Yaskawa INFORM job: FRONT_WELD_-90ST-1_5340.JBI

/JOB
//NAME FRONT_WELD_-90ST-1_5340
///FOLDERNAME 02-SKRZYNIE_JOBS
//POS
///NPOS 21,21,0,4,0,0
///TOOL 0
///POSTYPE PULSE
///PULSE
C00000=0,-52278,40443,0,6873,1
C00001=0,-52278,40443,0,6873,-1
C00002=0,-52278,40443,-5610,-49281,70968
C00003=0,-42686,23640,-7425,-34877,79161
C00004=14116,-58141,-26117,21696,-5351,66126
C00005=78387,-34691,-23344,93705,-44285,35747
C00006=74588,-16459,-14592,116746,-41260,23896
C00007=70798,-11760,-4995,114918,-37501,24909
C00008=60163,-19553,-11554,117597,-30554,22937
C00009=50151,-25103,-15872,121804,-24223,20236
C00010=32865,-30865,-19830,139529,-14643,10539
C00011=35290,-36639,-28855,139061,-17114,10894
C00012=3902,-39042,-32149,3317,17100,71988
C00013=3902,-39042,-32149,3317,17100,71988
C00014=3166,-35611,-25718,6481,14452,70496
C00015=-17642,-34526,-25309,42578,21356,51692
C00016=-28711,-32584,-24143,51084,27401,46743
C00017=-46420,-26852,-20499,57408,38357,42374
C00018=-48063,-35826,-27915,64657,37344,38904
C00019=-24039,-44019,6278,32369,22109,19464
C00020=0,-52278,40443,0,6873,-1
BC00000=801035
BC00001=820842
BC00002=820842
BC00003=949123
BC00004=997697
BC00005=1021293
BC00006=1027363
BC00007=1027363
BC00008=1027363
BC00009=1027363
BC00010=1027363
BC00011=1027363
BC00012=1027037
BC00013=1027037
BC00014=1027037
BC00015=1027039
BC00016=1027041
BC00017=1027043
BC00018=1027037
BC00019=924034
BC00020=820842
///POSTYPE BASE
///RECTAN
///RCONF 0,0,0,0,0,0,0,0,0,0,0,0,0,0,0,0,0,0,0,0,0,0,0,0
P00501=-2.026,0.009,3.534,0.0000,0.0000,0.0000
///RCONF 1,0,0,0,0,0,0,0,0,0,0,0,0,0,0,0,0,0,0,0,0,0,0,0
P00502=-2.023,0.001,1.732,0.0000,0.0000,0.0000
P00503=0.138,-0.044,1.539,0.0000,0.0000,0.0000
P00504=-0.309,-0.010,1.636,0.0000,0.0000,0.0000
//INST
///DATE 2024/08/01 10:17
///ATTR SC,RW
///GROUP1 RB1,BS1
NOP
MOVJ C00000 BC00000 VJ=50.00
MOVJ C00001 BC00001 VJ=50.00
MOVJ C00002 BC00002 VJ=50.00
MOVJ C00003 BC00003 VJ=50.00
MOVJ C00004 BC00004 VJ=50.00
MOVJ C00005 BC00005 VJ=50.00
'::::::::::::::::::::::::::::::::
'W56
'::::::::::::::::::::::::::::::::
MOVL C00006 BC00006 V=500.0
SFTON P0501
MACRO1 MJ#(0) ARGF14
MOVL C00007 BC00007 V=166.7 PL=0
ARCON
MOVC C00008 BC00008 V=9.5
SFTOF
SFTON P0502
MOVC C00009 BC00009 V=9.5
MOVC C00010 BC00010 V=9.5
ARCOF
MOVL C00011 BC00011 V=166.7
SFTOF
MOVL C00012 BC00012 V=166.7
'::::::::::::::::::::::::::::::::
'W21
'::::::::::::::::::::::::::::::::
MOVL C00013 BC00013 V=166.7
SFTON P0503
MACRO1 MJ#(0) ARGF14
MOVL C00014 BC00014 V=166.7 PL=0
ARCON
MOVL C00015 BC00015 V=9.5
SFTOF
SFTON P0504
MOVL C00016 BC00016 V=9.5
MOVL C00017 BC00017 V=9.5
ARCOF
MOVL C00018 BC00018 V=250.0
SFTOF
MOVJ C00019 BC00019 VJ=30.00
MOVJ C00020 BC00020 VJ=50.00
END
